FUNCTION_BLOCK FB_GetHttpConnectionParams
VAR_INPUT
	i_bExecute	: BOOL;
	i_sHttpUrl	: T_MaxString;
END_VAR
VAR_OUTPUT
	o_bError	: BOOL;
	o_nErrId	: UDINT;
	o_bReady	: BOOL;
	o_stHttpConnectionParams : ST_HTTP_Connection_Parameters;
END_VAR
VAR
	fbGetHostAddrByName		: FB_GetHostAddrByName;
	stHttpConnectionParams 	: ST_HTTP_Connection_Parameters;
	execute_R_TRIG			: R_TRIG;
	getHostAddrBusy_F_TRIG	: F_TRIG;
	bExecute				: BOOL;
	bUrlValid: BOOL;
	nState: INT := 10;
END_VAR



CASE nState OF
	
10: (* init *)
	nState := 20;
	
20:	(* Waiting for start *)
	
	IF i_bExecute THEN
		(* Reset *)
		o_bReady := FALSE;
		o_bError := FALSE;
		o_nErrId := 0;
		MEMSET(ADR(o_stHttpConnectionParams), 0, SIZEOF(o_stHttpConnectionParams));
		
		IF F_ParseHttpUrl(i_sHttpUrl, stHttpConnectionParams) THEN
			IF stHttpConnectionParams.sHostName <> 'localhost' THEN

				nState := 30;
			ELSE
				stHttpConnectionParams.sIpv4Address := '127.0.0.1';	
				o_stHttpConnectionParams := stHttpConnectionParams;
				o_bReady := TRUE;
				nState := 20;			
			END_IF
		ELSE 
			o_bError := TRUE;
		END_IF
	END_IF

30:	(* Waiting for ready *)

	fbGetHostAddrByName(
		sHostName	:= stHttpConnectionParams.sHostName,
		bExecute 	:= TRUE,
		tTimeout 	:= T#10S
	);
	
	IF fbGetHostAddrByName.bError THEN
		fbGetHostAddrByName(bExecute := FALSE);
		o_bError := TRUE;
		o_nErrId := fbGetHostAddrByName.nErrID;
		nState := 100;
	ELSIF NOT fbGetHostAddrByName.bBusy THEN
		fbGetHostAddrByName(bExecute := FALSE);
		stHttpConnectionParams.sIpv4Address := fbGetHostAddrByName.sAddr;
		o_stHttpConnectionParams := stHttpConnectionParams;
		o_bReady := TRUE;
		nState := 20;
	END_IF
	
100: (* Error state*)

	IF NOT i_bExecute THEN
		nState := 10;
	END_IF

END_CASE

END_FUNCTION_BLOCK

(* stored: Version 1.1.0.1, ProductVersion 3.1.4020.12
   POU FB_GetHttpConnectionParams: Id {3ccdec99-57cf-4a75-be13-c92fcaf8c943}, SpecialFunc None *)
